		tempLeg[0]:=legExtendRefPosCurling[i,0];tempLeg[1]:=legExtendRefPosCurling[i,1];tempLeg[2]:=legExtendRefPosCurling[i,2];
		tempRef[0]:=jntExtendRefPosCurling[i,0];tempRef[1]:=jntExtendRefPosCurling[i,1];tempRef[2]:=jntExtendRefPosCurling[i,2];
		GVL.legCtrl[i].InverseKinetics(tipPosition:=tempLeg , refPosLast:=tempRef , legIndex:=i , motorAngles=>tempJnt , isSingular=> );
		jntAngExtend[i,0]:=tempJnt[0];jntAngExtend[i,1]:=tempJnt[1];jntAngExtend[i,2]:=tempJnt[2];			
		
	END_FOR
	tipForceDesire:=tipForceDesireZeros;

END_IF

IF RecoveryFinished=FALSE THEN
	body_ref_pos:=body_ref_pos_enter;
	body_ref_ang:=body_ref_ang_enter;
	leg_ref_pos:=leg_ref_pos_enter;
	
	IF (gait_cycle-EnterRecoveryCount)<=(tRetract + tWait + tExtend) * gvl.sampleRate THEN //leg 0-2-4 recovery
		
		//force compensator****************************
		IF (gait_cycle-EnterRecoveryCount)<=fceLoadTime*gvl.sampleRate THEN
			tr  := UDINT_TO_LREAL(gait_cycle-EnterRecoveryCount) / gvl.sampleRate /fceLoadTime;
			fbGetPivot(tNow := tr, tTotal := 1.0, pivot => pvt);
			FOR i:=0 TO 5 DO
				FOR j:=0 TO 2 DO
					tipForceDesire[i,j]:=(1-pvt)*tipForceDesireZeros[i,j]+pvt*tipForceDesireGroupB[i,j];//group B add load
				END_FOR
			END_FOR
		ELSIF  (gait_cycle-EnterRecoveryCount)>LREAL_TO_UDINT((tRetract + tWait + tExtend-fceLoadTime)*gvl.sampleRate) AND  (gait_cycle-EnterRecoveryCount)<=LREAL_TO_UDINT((tRetract + tWait + tExtend) * gvl.sampleRate) THEN
			tr  := (UDINT_TO_LREAL (gait_cycle-EnterRecoveryCount) / gvl.sampleRate-(tRetract + tWait + tExtend-fceLoadTime) )/fceLoadTime;
			fbGetPivot(tNow := tr, tTotal := 1.0, pivot => pvt);
			FOR i:=0 TO 5 BY 2DO
				FOR j:=0 TO 2 DO
					//tipForceDesire[i,j]:=(1-pvt)*tipForceDesireZeros[i,j]+pvt*tipForceDesireGroupA[i,j];//group A add load
					tipForceDesire[i+1,j]:=(1-pvt)*tipForceDesireGroupB[i+1,j]+pvt*tipForceDesireZeros[i+1,j];//group B reduce load
				END_FOR
			END_FOR
		ELSE
		tipForceDesire:=tipForceDesireGroupB;
		END_IF
		//***********************************************
	
		IF gait_cycle-EnterRecoveryCount < tRetract * gvl.sampleRate THEN
			tTotal := tRetract;
			tNow   := UDINT_TO_LREAL(gait_cycle-EnterRecoveryCount) * 1.0 / DINT_TO_LREAL(gvl.sampleRate);
			jntPosBegin := RcJointPosStart;
			FOR i:=0 TO 5 BY 2 DO
				FOR j:=0 TO 2 DO
					jntPosEnd[i,j]:=jntAngRetract[i,j];
					jntPosEnd[i+1,j]:=RcJointPosStart[i+1,j];
				END_FOR
			END_FOR
		ELSIF gait_cycle-EnterRecoveryCount  < (tRetract + tWait) * gvl.sampleRate THEN
			tTotal := tWait;
			tNow   := UDINT_TO_LREAL(gait_cycle-EnterRecoveryCount) * 1.0 / DINT_TO_LREAL(gvl.sampleRate) - tRetract;
			FOR i:=0 TO 5 BY 2 DO
				FOR j:=0 TO 2 DO
					jntPosBegin[i,j]:=jntAngRetract[i,j];
					jntPosBegin[i+1,j]:=RcJointPosStart[i+1,j];
					jntPosEnd[i,j]:=jntAngRetract[i,j];
					jntPosEnd[i+1,j]:=RcJointPosStart[i+1,j];
				END_FOR
			END_FOR
		ELSE 
			tTotal := tExtend;
			tNow   := UDINT_TO_LREAL(gait_cycle-EnterRecoveryCount) * 1.0 / DINT_TO_LREAL(gvl.sampleRate) - tRetract - tWait;
			FOR i:=0 TO 5 BY 2 DO
				FOR j:=0 TO 2 DO
					jntPosBegin[i,j]:=jntAngRetract[i,j];
					jntPosBegin[i+1,j]:=RcJointPosStart[i+1,j];
					jntPosEnd[i,j]:=jntAngExtend[i,j];
					jntPosEnd[i+1,j]:=RcJointPosStart[i+1,j];
				END_FOR
			END_FOR	
		END_IF	
	ELSIF (gait_cycle-EnterRecoveryCount)<=2*(tRetract + tWait + tExtend) * gvl.sampleRate  THEN //leg 1-3-5 recovery

		//force compensator*******************
		IF (gait_cycle-EnterRecoveryCount)>LREAL_TO_UDINT((tRetract + tWait + tExtend)*gvl.sampleRate) AND (gait_cycle-EnterRecoveryCount)<=LREAL_TO_UDINT((tRetract + tWait + tExtend+fceLoadTime)* gvl.sampleRate) THEN
			tr  := (UDINT_TO_LREAL(gait_cycle-EnterRecoveryCount) / gvl.sampleRate-(tRetract + tWait + tExtend) )/fceLoadTime;
			fbGetPivot(tNow := tr, tTotal := 1.0, pivot => pvt);
			FOR i:=0 TO 5 BY 2 DO
				FOR j:=0 TO 2 DO
					tipForceDesire[i,j]:=(1-pvt)*tipForceDesireZeros[i,j]+pvt*tipForceDesireGroupA[i,j];//group A add load
					tipForceDesire[i+1,j]:=tipForceDesireZeros[i+1,j];//group B zeros load
				END_FOR
			END_FOR		
		ELSIF (gait_cycle-EnterRecoveryCount)>LREAL_TO_UDINT((2*(tRetract + tWait + tExtend)-fceLoadTime)*gvl.sampleRate) AND (gait_cycle-EnterRecoveryCount)<=LREAL_TO_UDINT(2*(tRetract + tWait + tExtend) * gvl.sampleRate) THEN
			tr  := (UDINT_TO_LREAL(gait_cycle-EnterRecoveryCount) / gvl.sampleRate-(2*(tRetract + tWait + tExtend)-fceLoadTime) )/fceLoadTime;
			fbGetPivot(tNow := tr, tTotal := 1.0, pivot => pvt);
			FOR i:=0 TO 5 BY 2DO
				FOR j:=0 TO 2 DO
					tipForceDesire[i,j]:=(1-pvt)*tipForceDesireGroupA[i,j]+pvt*tipForceDesireZeros[i,j];//group A reduce load
					tipForceDesire[i+1,j]:=tipForceDesireZeros[i+1,j];//group B zeros load
				END_FOR
			END_FOR	
		ELSE	
			tipForceDesire:=tipForceDesireGroupA;
		END_IF	
		//******************************************	

		
		IF gait_cycle-EnterRecoveryCount<=(2*tRetract + tWait + tExtend) * gvl.sampleRate THEN
			tTotal := tRetract;
			tNow   := UDINT_TO_LREAL(gait_cycle-EnterRecoveryCount) * 1.0 / DINT_TO_LREAL(gvl.sampleRate)-(tRetract + tWait + tExtend);
			FOR i:=0 TO 5 BY 2 DO
				FOR j:=0 TO 2 DO
					jntPosBegin[i,j]:=jntAngExtend[i,j];
					jntPosBegin[i+1,j]:=RcJointPosStart[i+1,j];
					jntPosEnd[i,j]:=jntAngExtend[i,j];
					jntPosEnd[i+1,j]:=jntAngRetract[i+1,j];
				END_FOR
			END_FOR			
		ELSIF gait_cycle-EnterRecoveryCount<=(2*tRetract + 2*tWait + tExtend) * gvl.sampleRate THEN
			tTotal := tWait;
			tNow   := UDINT_TO_LREAL(gait_cycle-EnterRecoveryCount) * 1.0 / DINT_TO_LREAL(gvl.sampleRate) - (2*tRetract + tWait + tExtend);
			FOR i:=0 TO 5 BY 2 DO
				FOR j:=0 TO 2 DO
					jntPosBegin[i,j]:=jntAngExtend[i,j];
					jntPosBegin[i+1,j]:=jntAngRetract[i+1,j];
					jntPosEnd[i,j]:=jntAngExtend[i,j];
					jntPosEnd[i+1,j]:=jntAngRetract[i+1,j];
				END_FOR
			END_FOR			
		ELSE
			tTotal := tExtend;
			tNow   := UDINT_TO_LREAL(gait_cycle-EnterRecoveryCount) * 1.0 / DINT_TO_LREAL(gvl.sampleRate) - (2*tRetract + 2*tWait + tExtend);
			FOR i:=0 TO 5 BY 2 DO
				FOR j:=0 TO 2 DO
					jntPosBegin[i,j]:=jntAngExtend[i,j];
					jntPosBegin[i+1,j]:=jntAngRetract[i+1,j];
					jntPosEnd[i,j]:=jntAngExtend[i,j];
					jntPosEnd[i+1,j]:=jntAngExtend[i+1,j];
				END_FOR
			END_FOR			
		END_IF
	ELSE
		tTotal := 100;
		tNow   := UDINT_TO_LREAL(gait_cycle-EnterRecoveryCount) * 1.0 / DINT_TO_LREAL(gvl.sampleRate) - 2*tRetract - 2*tWait - 2*tExtend;
		jntPosBegin :=jntAngExtend;
		jntPosEnd :=jntAngExtend;
		RecoveryFinished:=TRUE;
		tipForceDesire:=tipForceDesireZeros;
	END_IF
	getPivot(tNow := tNow, tTotal := tTotal, pivot => pivot, pivotDot => pivotDot);
	FOR i := 0 TO 5 DO
		FOR j := 0 TO 2 DO
			RcJointPosRef[i, j] := (1.0 - pivot) * jntPosBegin[i, j] + pivot * jntPosEnd[i, j];
		END_FOR
		tempJnt[0]:=RcJointPosRef[i,0];tempJnt[1]:=RcJointPosRef[i,1];tempJnt[2]:=RcJointPosRef[i,2];
		gvl.legCtrl[i].ForwardKinetics(motorAngles:=tempJnt , legIndex:=i , tipPosition=>Rc_PosWrtHip[i].data );
		fbRotMat(yaw := body_ref_ang_enter.data[2], pitch := body_ref_ang_enter.data[1],roll := body_ref_ang_enter.data[0], rm =>  Rb_target1 );
		temp.data[0]:=hip_pos[i,0];temp.data[1]:=hip_pos[i,1];temp.data[2]:=hip_pos[i,2];
		leg_ref_pos[i]:= VecAdd( MatMulVec(Rb_target1, VecAdd(temp,MatMulVec(Rleg[i],Rc_PosWrtHip[i]))),body_ref_pos);		
	END_FOR

END_IF
END_METHOD

METHOD PUBLIC TrjPlanning_SearchPedal : BOOL
VAR_INPUT
END_VAR
VAR
	tr: LREAL;
	i: INT;
	j: INT;
	Rb_target1: Mat3;
	temp: vec3;
	
	tipForceDesireLegA:	 ARRAY[0..5,0..2] OF LREAL:=[0,-100,0,
													 0,0,0,
													 0,0,0,
													 0,0,0,
													 0,0,0,
													 0,0,0];
	tipForceDesireLegF:	 ARRAY[0..5,0..2] OF LREAL:=[0,0,0,
													 0,0,0,
													 0,0,0,
													 0,0,0,
													 0,0,0,
													 0,-120,0];				
END_VAR
IF SearchPedalFinished=FALSE THEN
	IF SP_RBLegSearching=TRUE THEN
		SP_LBLegSearching:=FALSE;
		body_ref_pos:=body_ref_pos_enter;
		body_ref_ang:=body_ref_ang_enter;
		leg_ref_pos:=leg_ref_pos_enter;	
		IF (gait_cycle-SP_EnterSubSearchCount[0])<=SP_LiftLegTime*gvl.sampleRate THEN
			tr  := UDINT_TO_LREAL(gait_cycle - SP_EnterSubSearchCount[0]) / gvl.sampleRate / SP_LiftLegTime;
			fbGetPivot(tNow := tr, tTotal := 1.0, pivot => pvt);	
			SP_BPosRefWrtHip[0].data[0]:=SP_BPosStartWrtHip[0].data[0];
			SP_BPosRefWrtHip[0].data[1]:=(1-pvt)*SP_BPosStartWrtHip[0].data[1]+pvt*(SP_BPosStartWrtHip[0].data[1]+SP_LiftDistance);
			SP_BPosRefWrtHip[0].data[2]:=SP_BPosStartWrtHip[0].data[2];
			fbRotMat(yaw := body_ref_ang_enter.data[2], pitch := body_ref_ang_enter.data[1],roll := body_ref_ang_enter.data[0], rm =>  Rb_target1 );
			temp.data[0]:=hip_pos[0,0];temp.data[1]:=hip_pos[0,1];temp.data[2]:=hip_pos[0,2];
			leg_ref_pos[0]:= VecAdd( MatMulVec(Rb_target1, VecAdd(temp,MatMulVec(Rleg[0],SP_BPosRefWrtHip[0]))),body_ref_pos);	
			
			//force compensator
			tipForceTarget:=tipForceDesireLegF;
			IF (gait_cycle-SP_EnterSubSearchCount[0])<=LREAL_TO_UDINT(fceLoadTime*gvl.sampleRate) THEN
				tr  := (UDINT_TO_LREAL(gait_cycle-SP_EnterSubSearchCount[0]) / gvl.sampleRate)/ fceLoadTime;
				fbGetPivot(tNow := tr, tTotal := 1.0, pivot => pvt);
				FOR i:=0 TO 5 DO
					FOR j:=0 TO 2 DO
						tipForceDesire[i,j]:=(1-pvt)*tipForceDesireZeros[i,j]+pvt*tipForceTarget[i,j];
					END_FOR
				END_FOR
			END_IF
			
		ELSIF (gait_cycle-SP_EnterSubSearchCount[0])<=(SP_LiftLegTime+SP_SearchTime)*gvl.sampleRate AND  SP_BLegSearchFinished[0]=FALSE THEN
			tr  := (UDINT_TO_LREAL(gait_cycle - SP_EnterSubSearchCount[0]) / gvl.sampleRate -SP_LiftLegTime)/ SP_SearchTime;
			fbGetPivot(tNow := tr, tTotal := 1.0, pivot => pvt);	
			SP_BPosRefWrtHip[0].data[0]:=(1-pvt)*SP_BPosStartWrtHip[0].data[0]+pvt*(SP_BPosStartWrtHip[0].data[0]-SP_SearchDistance);		
			SP_BPosRefWrtHip[0].data[1]:=SP_BPosStartWrtHip[0].data[1]+SP_LiftDistance;
			SP_BPosRefWrtHip[0].data[2]:=SP_BPosStartWrtHip[0].data[2];
			IF isPedal(0)=TRUE AND  SP_BLegSearchFinished[0]=FALSE THEN
				SP_BLegSearchFinished[0]:=TRUE;
				SP_EnterSubSearchDecreaseCount[0]:=gait_cycle;
				FOR j:=0 TO 2 DO
					SP_BPosLockWrtHip[0].data[j]:=SP_BPosRefWrtHip[0].data[j];
				END_FOR			
			END_IF
			IF (gait_cycle-SP_EnterSubSearchCount[0])=LREAL_TO_UDINT((SP_LiftLegTime+SP_SearchTime)*gvl.sampleRate) AND SP_BLegSearchFinished[0]=FALSE THEN
				SP_BLegSearchFinished[0]:=TRUE;
				SP_EnterSubSearchDecreaseCount[0]:=gait_cycle;
				FOR j:=0 TO 2 DO
					SP_BPosLockWrtHip[0].data[j]:=SP_BPosRefWrtHip[0].data[j];
				END_FOR	
			END_IF

			fbRotMat(yaw := body_ref_ang_enter.data[2], pitch := body_ref_ang_enter.data[1],roll := body_ref_ang_enter.data[0], rm =>  Rb_target1 );
			temp.data[0]:=hip_pos[0,0];temp.data[1]:=hip_pos[0,1];temp.data[2]:=hip_pos[0,2];
			leg_ref_pos[0]:= VecAdd( MatMulVec(Rb_target1, VecAdd(temp,MatMulVec(Rleg[0],SP_BPosRefWrtHip[0]))),body_ref_pos);	
			
		ELSIF  SP_BLegSearchFinished[0]=TRUE AND (gait_cycle-SP_EnterSubSearchDecreaseCount[0])<=SP_LiftLegTime*gvl.sampleRate THEN
			tr  := UDINT_TO_LREAL(gait_cycle - SP_EnterSubSearchDecreaseCount[0]) / gvl.sampleRate / SP_LiftLegTime;
			fbGetPivot(tNow := tr, tTotal := 1.0, pivot => pvt);
			SP_BPosRefWrtHip[0].data[0]:=SP_BPosLockWrtHip[0].data[0];	
			SP_BPosRefWrtHip[0].data[1]:=(1-pvt)*SP_BPosLockWrtHip[0].data[1]+pvt*(SP_BPosLockWrtHip[0].data[1]-SP_LiftDistance);
			SP_BPosRefWrtHip[0].data[2]:=SP_BPosLockWrtHip[0].data[2];	
			
			fbRotMat(yaw := body_ref_ang_enter.data[2], pitch := body_ref_ang_enter.data[1],roll := body_ref_ang_enter.data[0], rm =>  Rb_target1 );
			temp.data[0]:=hip_pos[0,0];temp.data[1]:=hip_pos[0,1];temp.data[2]:=hip_pos[0,2];
			leg_ref_pos[0]:= VecAdd( MatMulVec(Rb_target1, VecAdd(temp,MatMulVec(Rleg[0],SP_BPosRefWrtHip[0]))),body_ref_pos);	
			IF (gait_cycle-SP_EnterSubSearchDecreaseCount[0])=LREAL_TO_UDINT( SP_LiftLegTime*gvl.sampleRate) THEN
				body_ref_pos_enter:=body_ref_pos;
				body_ref_ang_enter:=body_ref_ang;
				leg_ref_pos_enter:=leg_ref_pos;	
			END_IF	
			
			//force compensator
			tipForceTarget:=tipForceDesireLegF;
			IF (gait_cycle-SP_EnterSubSearchDecreaseCount[0])>LREAL_TO_UDINT((SP_LiftLegTime-fceLoadTime)*gvl.sampleRate)THEN
				tr  := (UDINT_TO_LREAL(gait_cycle-SP_EnterSubSearchDecreaseCount[0]) / gvl.sampleRate-(SP_LiftLegTime-fceLoadTime) )/ fceLoadTime;
				fbGetPivot(tNow := tr, tTotal := 1.0, pivot => pvt);
				FOR i:=0 TO 5 DO
					FOR j:=0 TO 2 DO
						tipForceDesire[i,j]:=(1-pvt)*tipForceTarget[i,j]+pvt*tipForceDesireZeros[i,j];
					END_FOR
				END_FOR
			END_IF
	
		ELSE
			SP_RBLegSearching:=FALSE;
			SP_LBLegSearching:=TRUE;
			SP_EnterSubSearchCount[1]:=gait_cycle;			
		END_IF
	END_IF
	
	IF SP_LBLegSearching=TRUE THEN
		SP_RBLegSearching:=FALSE;
		body_ref_pos:=body_ref_pos_enter;
		body_ref_ang:=body_ref_ang_enter;
		leg_ref_pos:=leg_ref_pos_enter;	
		IF (gait_cycle-SP_EnterSubSearchCount[1])<=SP_LiftLegTime*gvl.sampleRate THEN
			tr  := UDINT_TO_LREAL(gait_cycle - SP_EnterSubSearchCount[1]) / gvl.sampleRate / SP_LiftLegTime;
			fbGetPivot(tNow := tr, tTotal := 1.0, pivot => pvt);	
			SP_BPosRefWrtHip[1].data[0]:=SP_BPosStartWrtHip[1].data[0];
			SP_BPosRefWrtHip[1].data[1]:=(1-pvt)*SP_BPosStartWrtHip[1].data[1]+pvt*(SP_BPosStartWrtHip[1].data[1]+SP_LiftDistance);
			SP_BPosRefWrtHip[1].data[2]:=SP_BPosStartWrtHip[1].data[2];
			fbRotMat(yaw := body_ref_ang_enter.data[2], pitch := body_ref_ang_enter.data[1],roll := body_ref_ang_enter.data[0], rm =>  Rb_target1 );
			temp.data[0]:=hip_pos[5,0];temp.data[1]:=hip_pos[5,1];temp.data[2]:=hip_pos[5,2];
			leg_ref_pos[5]:= VecAdd( MatMulVec(Rb_target1, VecAdd(temp,MatMulVec(Rleg[5],SP_BPosRefWrtHip[1]))),body_ref_pos);	
			
			//force compensator
			tipForceTarget:=tipForceDesireLegA;
			IF (gait_cycle-SP_EnterSubSearchCount[1])<=LREAL_TO_UDINT(fceLoadTime*gvl.sampleRate) THEN
				tr  := (UDINT_TO_LREAL(gait_cycle-SP_EnterSubSearchCount[1]) / gvl.sampleRate)/ fceLoadTime;
				fbGetPivot(tNow := tr, tTotal := 1.0, pivot => pvt);
				FOR i:=0 TO 5 DO
					FOR j:=0 TO 2 DO
						tipForceDesire[i,j]:=(1-pvt)*tipForceDesireZeros[i,j]+pvt*tipForceTarget[i,j];
					END_FOR
				END_FOR
			END_IF
			
		ELSIF (gait_cycle-SP_EnterSubSearchCount[1])<=(SP_LiftLegTime+SP_SearchTime)*gvl.sampleRate AND  SP_BLegSearchFinished[1]=FALSE THEN
			tr  := (UDINT_TO_LREAL(gait_cycle - SP_EnterSubSearchCount[1]) / gvl.sampleRate -SP_LiftLegTime)/ SP_SearchTime;
			fbGetPivot(tNow := tr, tTotal := 1.0, pivot => pvt);	
			SP_BPosRefWrtHip[1].data[0]:=(1-pvt)*SP_BPosStartWrtHip[1].data[0]+pvt*(SP_BPosStartWrtHip[1].data[0]-SP_SearchDistance);		
			SP_BPosRefWrtHip[1].data[1]:=SP_BPosStartWrtHip[1].data[1]+SP_LiftDistance;
			SP_BPosRefWrtHip[1].data[2]:=SP_BPosStartWrtHip[1].data[2];
			IF isPedal(5)=TRUE AND  SP_BLegSearchFinished[1]=FALSE THEN
				SP_BLegSearchFinished[1]:=TRUE;
				SP_EnterSubSearchDecreaseCount[1]:=gait_cycle;
				FOR j:=0 TO 2 DO
					SP_BPosLockWrtHip[1].data[j]:=SP_BPosRefWrtHip[1].data[j];
				END_FOR			
			END_IF
			IF (gait_cycle-SP_EnterSubSearchCount[1])=LREAL_TO_UDINT((SP_LiftLegTime+SP_SearchTime)*gvl.sampleRate) AND SP_BLegSearchFinished[1]=FALSE THEN
				SP_BLegSearchFinished[1]:=TRUE;
				SP_EnterSubSearchDecreaseCount[1]:=gait_cycle;
				FOR j:=0 TO 2 DO
					SP_BPosLockWrtHip[1].data[j]:=SP_BPosRefWrtHip[1].data[j];
				END_FOR	
			END_IF

			fbRotMat(yaw := body_ref_ang_enter.data[2], pitch := body_ref_ang_enter.data[1],roll := body_ref_ang_enter.data[0], rm =>  Rb_target1 );
			temp.data[0]:=hip_pos[5,0];temp.data[1]:=hip_pos[5,1];temp.data[2]:=hip_pos[5,2];
			leg_ref_pos[5]:= VecAdd( MatMulVec(Rb_target1, VecAdd(temp,MatMulVec(Rleg[5],SP_BPosRefWrtHip[1]))),body_ref_pos);	
			
		ELSIF  SP_BLegSearchFinished[1]=TRUE AND (gait_cycle-SP_EnterSubSearchDecreaseCount[1])<=SP_LiftLegTime*gvl.sampleRate THEN
			tr  := UDINT_TO_LREAL(gait_cycle - SP_EnterSubSearchDecreaseCount[1]) / gvl.sampleRate / SP_LiftLegTime;
			fbGetPivot(tNow := tr, tTotal := 1.0, pivot => pvt);
			SP_BPosRefWrtHip[1].data[0]:=SP_BPosLockWrtHip[1].data[0];	
			SP_BPosRefWrtHip[1].data[1]:=(1-pvt)*SP_BPosLockWrtHip[1].data[1]+pvt*(SP_BPosLockWrtHip[1].data[1]-SP_LiftDistance);
			SP_BPosRefWrtHip[1].data[2]:=SP_BPosLockWrtHip[1].data[2];	
			
			fbRotMat(yaw := body_ref_ang_enter.data[2], pitch := body_ref_ang_enter.data[1],roll := body_ref_ang_enter.data[0], rm =>  Rb_target1 );
			temp.data[0]:=hip_pos[5,0];temp.data[1]:=hip_pos[5,1];temp.data[2]:=hip_pos[5,2];
			leg_ref_pos[5]:= VecAdd( MatMulVec(Rb_target1, VecAdd(temp,MatMulVec(Rleg[5],SP_BPosRefWrtHip[1]))),body_ref_pos);	
			IF (gait_cycle-SP_EnterSubSearchDecreaseCount[1])=LREAL_TO_UDINT( SP_LiftLegTime*gvl.sampleRate) THEN
				body_ref_pos_enter:=body_ref_pos;
				body_ref_ang_enter:=body_ref_ang;
				leg_ref_pos_enter:=leg_ref_pos;	
			END_IF	
			
			//force compensator
			tipForceTarget:=tipForceDesireLegA;
			IF (gait_cycle-SP_EnterSubSearchDecreaseCount[1])>LREAL_TO_UDINT((SP_LiftLegTime-fceLoadTime)*gvl.sampleRate)THEN
				tr  := (UDINT_TO_LREAL(gait_cycle-SP_EnterSubSearchDecreaseCount[1]) / gvl.sampleRate-(SP_LiftLegTime-fceLoadTime) )/ fceLoadTime;
				fbGetPivot(tNow := tr, tTotal := 1.0, pivot => pvt);
				FOR i:=0 TO 5 DO
					FOR j:=0 TO 2 DO
						tipForceDesire[i,j]:=(1-pvt)*tipForceTarget[i,j]+pvt*tipForceDesireZeros[i,j];
					END_FOR
				END_FOR
			END_IF			
			
		ELSE
			SP_RBLegSearching:=FALSE;
			SP_LBLegSearching:=FALSE;	
			SearchPedalFinished:=TRUE;	
			tipForceDesire:=tipForceDesireZeros;
		END_IF
	END_IF	
END_IF
END_METHOD

METHOD PUBLIC TrjPlanning_Slide : BOOL
VAR_INPUT
END_VAR
IF SlideFinished=FALSE THEN
	body_ref_pos:=body_ref_pos_enter;
	body_ref_ang:=body_ref_ang_enter;
	leg_ref_pos:=leg_ref_pos_enter;

END_IF

//***********tuning***************************
IF SlideFinished=FALSE AND (gait_cycle-EnterSlideCount)>=LREAL_TO_UDINT(slideTime*gvl.sampleRate) THEN
	RequirePushReleaseBall:=TRUE;
END_IF

//*************end-tuning********************



IF SlideFinished=FALSE AND RequirePushReleaseBall=TRUE THEN
	SlideFinished:=TRUE;
END_IF
END_METHOD

METHOD PUBLIC TrjPlanning_SpeedDown : BOOL
VAR_INPUT
END_VAR

VAR
	tr: LREAL;
	i: INT;
	SpeedDown_MPosTarget:ARRAY[0..1,0..2] OF LREAL:=[-0.0141,-0.1797,-0.1246,
                                                        -0.0141,-0.1797,0.1246];
	SpeedDown_MJntTargetRef:ARRAY[0..1,0..2] OF LREAL:=[0,331.45*pi/180,-144*pi/180,
                                                     0,331.45*pi/180,-144*pi/180];
	j: INT;
	Rb_target1: Mat3;
	temp: vec3;
	tempLeg:ARRAY [0..2] OF LREAL;
	tempJnt:ARRAY [0..2] OF LREAL;
	tempRef:ARRAY [0..2] OF LREAL;
END_VAR
IF (gait_cycle-EnterSpeedDownCount)=1 THEN
	FOR i:=0 TO 1 DO
		tempLeg[0]:=SpeedDown_MPosTarget[i,0];tempLeg[1]:=SpeedDown_MPosTarget[i,1];tempLeg[2]:=SpeedDown_MPosTarget[i,2];
		tempRef[0]:=SpeedDown_MJntTargetRef[i,0];tempRef[1]:=SpeedDown_MJntTargetRef[i,1];tempRef[2]:=SpeedDown_MJntTargetRef[i,2];
		GVL.legCtrl[Mapping14[i]].InverseKinetics(tipPosition:=tempLeg , refPosLast:=tempRef , legIndex:=Mapping14[i] , motorAngles=>tempJnt , isSingular=> );
		SpeedDown_MJntTarget[i,0]:=tempJnt[0];SpeedDown_MJntTarget[i,1]:=tempJnt[1];SpeedDown_MJntTarget[i,2]:=tempJnt[2];		
	END_FOR
END_IF

IF SpeedDownFinished=FALSE THEN
	IF gait_cycle-EnterSpeedDownCount<=SpeedDownTime*gvl.sampleRate THEN
		body_ref_pos:=body_ref_pos_enter;
		body_ref_ang:=body_ref_ang_enter;
		leg_ref_pos:=leg_ref_pos_enter;
		tr  := UDINT_TO_LREAL(gait_cycle - EnterSpeedDownCount) / gvl.sampleRate / SpeedDownTime;
		fbGetPivot(tNow := tr, tTotal := 1.0, pivot => pvt);
		FOR i:=0 TO 1 DO
			FOR j:=0 TO 2 DO
				SpeedDown_MJntRef[i].data[j]:=(1-pvt)*SpeedDown_MJntStart[i].data[j]+pvt*SpeedDown_MJntTarget[i,j];
			END_FOR
			gvl.legCtrl[Mapping14[i]].ForwardKinetics(motorAngles:=SpeedDown_MJntRef[i].data , legIndex:=Mapping14[i] , tipPosition=>SpeedDown_MPosWrtHip[i].data );
			fbRotMat(yaw := body_ref_ang_enter.data[2], pitch := body_ref_ang_enter.data[1],roll := body_ref_ang_enter.data[0], rm =>  Rb_target1 );
			temp.data[0]:=hip_pos[Mapping14[i],0];temp.data[1]:=hip_pos[Mapping14[i],1];temp.data[2]:=hip_pos[Mapping14[i],2];
			leg_ref_pos[Mapping14[i]]:= VecAdd( MatMulVec(Rb_target1, VecAdd(temp,MatMulVec(Rleg[Mapping14[i]],SpeedDown_MPosWrtHip[i]))),body_ref_pos);
			
			leg_ref_pos[Mapping05[i]].data[2]:=(1-pvt)*leg_ref_pos_enter[Mapping05[i]].data[2]+pvt*(leg_ref_pos_enter[Mapping05[i]].data[2]-Distance_y_DS-0.005);
		END_FOR
	ELSE
		SpeedDownFinished:=TRUE;
	END_IF
	
	IF gait_cycle-EnterSpeedDownCount=1 THEN
		GVL.jogVelocity[18]:=0;
		GVL.jogVelocity[19]:=0;
		gvl.jogStopButton[18]:=TRUE;
		gvl.jogStopButton[19]:=TRUE;
		gvl.motorDrive[j].SetTrgVel(0);
	END_IF
END_IF
END_METHOD

METHOD PUBLIC TrjPlanning_SpeedUp : BOOL
VAR_INPUT
END_VAR

VAR
	invalid: LREAL;
	Rb_target1: Mat3;
	i: INT;
	tr: LREAL;
	temp: VEC3;
	
	
	tipForceDesireLegAF:	 ARRAY[0..5,0..2] OF LREAL:=[0,-30,0,
													 0,0,0,
													 0,0,0,
													 0,0,0,
													 0,0,0,
													 0,-30,0];
	j: INT;
END_VAR
IF SpeedUpSubState=SpeedUpAS AND (gait_cycle-EnterSpeedUpASCount)=LREAL_TO_UDINT(Time_AS*gvl.sampleRate) THEN
	SpeedUpSubState:=SpeedUpCS;
	EnterSpeedUpCSCount:=gait_cycle;
	body_ref_pos_enter :=body_ref_pos;
	body_ref_ang_enter:=body_ref_ang;
	leg_ref_pos_enter := leg_ref_pos;
	
ELSIF SpeedUpSubState=SpeedUpCS AND gait_cycle-EnterSpeedUpCSCount=LREAL_TO_UDINT(Time_CS*gvl.sampleRate) THEN
	SpeedUpSubState:=SpeedUpDS;
	EnterSpeedUpDSCount:=gait_cycle;
	body_ref_pos_enter :=body_ref_pos;
	body_ref_ang_enter:=body_ref_ang;
	leg_ref_pos_enter := leg_ref_pos;
ELSIF SpeedUpSubState=SpeedUpDS AND gait_cycle-EnterSpeedUpDSCount=LREAL_TO_UDINT(Time_DS*gvl.sampleRate) THEN
	SpeedUpSubState:=SpeedUpSS;
	EnterSpeedUpSPCount:=gait_cycle;
	body_ref_pos_enter :=body_ref_pos;
	body_ref_ang_enter:=body_ref_ang;
	leg_ref_pos_enter := leg_ref_pos;
	SpeedUpFinished:=TRUE;
	tipForceDesire:=tipForceDesireZeros;
	RequireSlide:=TRUE;
END_IF

body_ref_pos:=body_ref_pos_enter;
body_ref_ang:=body_ref_ang_enter;
leg_ref_pos:=leg_ref_pos_enter;

IF SpeedUpSubState=SpeedUpAS AND gait_cycle-EnterSpeedUpASCount<=Time_AS*gvl.sampleRate THEN
	fbHermitInterpolation(t0:=EnterSpeedUpASCount*delta_t , T:=Time_AS , y0:=0 , 
		y1:=Distance_x_AS , v0:=0 , v1:=target_vel , tNow:=gait_cycle* delta_t, 
		y=> body_ref_pos_wrt_body.data[0], v=>invalid );	
	body_ref_pos_wrt_body.data[1]:=0;body_ref_pos_wrt_body.data[2]:=0;
	fbRotMat(yaw := body_ref_ang_enter.data[2], pitch := body_ref_ang_enter.data[1],roll := body_ref_ang_enter.data[0], rm =>  Rb_target1 );
	body_ref_pos:=VecAdd(body_ref_pos_enter,MatMulVec(Rb_target1,body_ref_pos_wrt_body));
	
	//force compensator
	tipForceTarget:=tipForceDesireLegAF;
	IF (gait_cycle-EnterSpeedUpASCount)<=fceLoadTime*gvl.sampleRate THEN
		tr  := UDINT_TO_LREAL(gait_cycle-EnterSpeedUpASCount) / gvl.sampleRate / fceLoadTime;
		fbGetPivot(tNow := tr, tTotal := 1.0, pivot => pvt);
		FOR i:=0 TO 5 DO
			FOR j:=0 TO 2 DO
				tipForceDesire[i,j]:=(1-pvt)*tipForceDesireZeros[i,j]+pvt*tipForceTarget[i,j];
			END_FOR
		END_FOR	
	END_IF
	
END_IF
	//force compensator
	tipForceTarget:=tipForceDesireLegAF;
	IF (gait_cycle-EnterSpeedUpASCount)>(Time_AS+Time_CS-fceLoadTime)*gvl.sampleRate AND (gait_cycle-EnterSpeedUpASCount)<=(Time_AS+Time_CS)*gvl.sampleRate THEN
		tr  := (UDINT_TO_LREAL(gait_cycle-EnterSpeedUpASCount) / gvl.sampleRate- (Time_AS+Time_CS-fceLoadTime))/ fceLoadTime;
		fbGetPivot(tNow := tr, tTotal := 1.0, pivot => pvt);
		FOR i:=0 TO 5 DO
			FOR j:=0 TO 2 DO
				tipForceDesire[i,j]:=(1-pvt)*tipForceTarget[i,j]+pvt*tipForceDesireZeros[i,j];
			END_FOR
		END_FOR	
	END_IF

IF SpeedUpSubState=SpeedUpCS AND gait_cycle-EnterSpeedUpCSCount<=Time_CS*gvl.sampleRate THEN
	fbHermitInterpolation(t0:=EnterSpeedUpCSCount*delta_t , T:=Time_CS , y0:=0 , 
		y1:=target_vel*Time_CS , v0:=target_vel , v1:=target_vel , tNow:=gait_cycle* delta_t, 
		y=> body_ref_pos_wrt_body.data[0], v=>invalid );
	body_ref_pos_wrt_body.data[1]:=0;body_ref_pos_wrt_body.data[2]:=0;
	fbRotMat(yaw := body_ref_ang_enter.data[2], pitch := body_ref_ang_enter.data[1],roll := body_ref_ang_enter.data[0], rm =>  Rb_target1 );
	body_ref_pos:=VecAdd(body_ref_pos_enter,MatMulVec(Rb_target1,body_ref_pos_wrt_body));
END_IF
IF SpeedUpSubState=SpeedUpDS AND gait_cycle-EnterSpeedUpDSCount<=Time_DS*gvl.sampleRate THEN
	fbHermitInterpolation(t0:=EnterSpeedUpDSCount*delta_t , T:=Time_DS , y0:=0 , 
		y1:=Distance_x_DS , v0:=target_vel , v1:=0 , tNow:=gait_cycle* delta_t, 
		y=> body_ref_pos_wrt_body.data[0], v=>invalid );
	body_ref_pos_wrt_body.data[1]:=0;body_ref_pos_wrt_body.data[2]:=0;
	
	fbRotMat(yaw := body_ref_ang_enter.data[2], pitch := body_ref_ang_enter.data[1],roll := body_ref_ang_enter.data[0], rm =>  Rb_target1 );
	body_ref_pos:=VecAdd(body_ref_pos_enter,MatMulVec(Rb_target1,body_ref_pos_wrt_body));
	
	tr  := UDINT_TO_LREAL(gait_cycle - EnterSpeedUpDSCount) / gvl.sampleRate / Time_DS;
	fbGetPivot(tNow := tr, tTotal := 1.0, pivot => pvt);
	FOR i:=0 TO 1 DO
		leg_ref_pos[Mapping05[i]].data[2]:=(1-pvt)*leg_ref_pos_enter[Mapping05[i]].data[2]+pvt*(leg_ref_pos_enter[Mapping05[i]].data[2]+Distance_y_DS);
	END_FOR
	
END_IF
IF SpeedUpSubState=SpeedUpAS OR SpeedUpSubState=SpeedUpCS OR SpeedUpSubState=SpeedUpDS THEN
	FOR i:=0 TO 1 DO
		gvl.legCtrl[Mapping14[i]].ForwardKinetics(motorAngles:=SpeedUp_MJntRef[i].data , legIndex:=Mapping14[i] , tipPosition=>SpeedUp_MPosWrtHip[i].data );
		gvl.legCtrl[Mapping23[i]].ForwardKinetics(motorAngles:=SpeedUp_FJntRef[i].data , legIndex:=Mapping23[i] , tipPosition=>SpeedUp_FPosWrtHip[i].data );
		fbRotMat(yaw := body_ref_ang_enter.data[2], pitch := body_ref_ang_enter.data[1],roll := body_ref_ang_enter.data[0], rm =>  Rb_target1 );
		temp.data[0]:=hip_pos[Mapping14[i],0];temp.data[1]:=hip_pos[Mapping14[i],1];temp.data[2]:=hip_pos[Mapping14[i],2];
		leg_ref_pos[Mapping14[i]]:= VecAdd( MatMulVec(Rb_target1, VecAdd(temp,MatMulVec(Rleg[Mapping14[i]],SpeedUp_MPosWrtHip[i]))),body_ref_pos);
		temp.data[0]:=hip_pos[Mapping23[i],0];temp.data[1]:=hip_pos[Mapping23[i],1];temp.data[2]:=hip_pos[Mapping23[i],2];
		leg_ref_pos[Mapping23[i]]:= VecAdd( MatMulVec(Rb_target1, VecAdd(temp,MatMulVec(Rleg[Mapping23[i]],SpeedUp_FPosWrtHip[i]))),body_ref_pos);
	END_FOR
END_IF
END_METHOD

METHOD PUBLIC TrjPlanning_StoneRot : BOOL
VAR_INPUT
END_VAR
VAR
	(*StoneRot_FJntTarget:ARRAY[0..1,0..2] OF LREAL:=[-90*pi/180,524*pi/180,-190*pi/180,
                                                     90*pi/180,524*pi/180,-190*pi/180];*)
													 
	(*StoneRot_FJntTarget:ARRAY[0..1,0..2] OF LREAL:=[-90*pi/180,165*pi/180,(-190+360)*pi/180,
                                                     90*pi/180,165*pi/180,(-190+360)*pi/180];	//164 lose,165T 170S lose;*)
	StoneRot_FJntTarget:ARRAY[0..1,0..2] OF LREAL:=[-90*pi/180,167*pi/180,(171)*pi/180,
                                                     90*pi/180,167*pi/180,(171)*pi/180];	//164 lose,166T 168S passive wheels colide;												 
	tr: LREAL;
	i: INT;
	Rb_target1: Mat3;	
	temp:vec3;										 
	j: INT;
	noPlanning: BOOL;
END_VAR
//*****************************test trajectory*****************************************

	FOR i:=0 TO 1 DO
		(*IF SetColide=TRUE THEN
			gvl.tipActualFce[Mapping23[i],2]:=100;
		END_IF	*)
		(*IF(gait_cycle-EnterStoneRotCount)=0.5*StoneGripTime*gvl.sampleRate THEN
			gvl.tipActualFce[Mapping23[i],2]:=100;
		END_IF *)
		noPlanning:=TRUE;
	END_FOR
	

//**********************************end************************************************	

(*FOR i:=0 TO 1 DO
	IF StoneRotSubState[i]=FALSE AND isStone(Mapping23[i]) THEN
		StoneRotSubState[i]:=TRUE;
		leg_ref_pos_enter[Mapping23[i]]:=leg_ref_pos[Mapping23[i]];
	END_IF
END_FOR*)

IF (StoneRotSubState[0]=FALSE OR StoneRotSubState[1]=FALSE) AND (gait_cycle-EnterStoneRotCount)=LREAL_TO_UDINT(StoneGripTime*gvl.sampleRate) THEN
	StoneRotSubState[0]:=TRUE;
	StoneRotSubState[1]:=TRUE;
	leg_ref_pos_enter[Mapping23[0]]:=leg_ref_pos[Mapping23[0]];
	leg_ref_pos_enter[Mapping23[1]]:=leg_ref_pos[Mapping23[1]];
END_IF
	
body_ref_pos:=body_ref_pos_enter;
body_ref_ang:=body_ref_ang_enter;
leg_ref_pos:=leg_ref_pos_enter;


	IF (gait_cycle-EnterStoneRotCount)<=StoneGripTime*gvl.sampleRate THEN
		FOR i:=0 TO 1 DO
			IF StoneRotSubState[i]=FALSE THEN
			tr  := UDINT_TO_LREAL(gait_cycle - EnterStoneRotCount) / gvl.sampleRate /StoneGripTime;
			fbGetPivot(tNow := tr, tTotal := 1.0, pivot => pvt);
			FOR j:=0 TO 2 DO
				StoneRot_FJntRef[i].data[j]:=(1-pvt)*StoneRot_FJntStart[i].data[j]+pvt*(StoneRot_FJntTarget[i,j]);
			END_FOR
			gvl.legCtrl[Mapping23[i]].ForwardKinetics(motorAngles:=StoneRot_FJntRef[i].data , legIndex:=Mapping23[i] , tipPosition=>StoneRot_FPosWrtHip[i].data );
			fbRotMat(yaw := body_ref_ang_enter.data[2], pitch := body_ref_ang_enter.data[1],roll := body_ref_ang_enter.data[0], rm =>  Rb_target1 );
			temp.data[0]:=hip_pos[Mapping23[i],0];temp.data[1]:=hip_pos[Mapping23[i],1];temp.data[2]:=hip_pos[Mapping23[i],2];
			leg_ref_pos[Mapping23[i]]:= VecAdd( MatMulVec(Rb_target1, VecAdd(temp,MatMulVec(Rleg[Mapping23[i]],StoneRot_FPosWrtHip[i]))),body_ref_pos);
			END_IF
		END_FOR
	ELSE
		noPlanning:=TRUE;
	END_IF

IF (gait_cycle-EnterStoneRotCount)>StoneGripTime*gvl.sampleRate  THEN
		stone_rot_vel:=GVL.stone_rot_vel/60*2*pi;
		GVL.jogVelocity[18]:=stone_rot_vel;
		GVL.jogVelocity[19]:=-stone_rot_vel;
		FOR j:=18 TO 19 DO
			gvl.motorDrive[j].SetTrgVel(GVL.jogVelocity[j]);
			IF gvl.motorDrive[j].cvSetVel = GVL.jogVelocity[j] THEN
				gvl.jogButton[j]:=FALSE;
			ELSE
				gvl.jogButton[j]:=TRUE;
			END_IF
		END_FOR
END_IF

IF StoneRotFinished=FALSE AND (gait_cycle-EnterStoneRotCount)>=(StoneGripTime+StoneRotTime)*gvl.sampleRate THEN
	StoneRotFinished:=TRUE;
END_IF
END_METHOD

END_FUNCTION_BLOCK

(* stored: Version 1.1.0.1, ProductVersion 3.1.4024.2
   POU CurlingGaitFromSlip: Id {60870fbe-9372-4644-8201-6ee4a114d2cf}, SpecialFunc None
   Method DoPlanning: Id {a526c105-864a-4ef3-a646-bb7632c42b5f}
   Method Initialize: Id {9bdfb3b6-4c18-49e5-bc86-7a870e5fcc33}
   Method isPedal: Id {33785039-937e-483a-8149-9a6f9589866a}
   Method isStone: Id {3828978a-85ac-4eb4-8168-c31866fd1ac4}
   Method SetTargetValue: Id {e1935ec6-c32b-41cc-a62d-b61459b5fd30}
   Method StateMachine: Id {5ef4ea9d-f719-4140-9cda-9aefc2e8dc7a}
   Method TrjPlanning: Id {33080927-9d47-4eee-921a-6bb8a64b1112}
   Method TrjPlanning_AddHeight: Id {acb813a6-b8d3-446e-a4d2-e1b9c2cdd5b4}
   Method TrjPlanning_ArmControl: Id {99fa43a9-ec94-415c-9cd9-37ff750f7e87}
   Method TrjPlanning_BLegPosAdjust: Id {3093e979-b721-4bdb-95bd-ab44a7107aa5}
   Method TrjPlanning_BLegRecovery: Id {cd829a26-9eb0-4fd9-96d1-940c236395fe}
   Method TrjPlanning_BodyPosAdjust: Id {7f0117a2-a706-4595-9d97-7df79ab3b366}
   Method TrjPlanning_FlegRotB: Id {c1a7410f-1fb6-41d5-8519-4751dfebdb87}
   Method TrjPlanning_LiftMleg: Id {a543d1fd-a688-4e1e-a9a0-947506f19caf}
   Method TrjPlanning_MlegRollA: Id {bfb227bd-ca7c-4e4b-92fd-b1a2b93a0523}
   Method TrjPlanning_MlegRollB: Id {76260543-839c-4ac6-a04d-6f8340937b67}
   Method TrjPlanning_MlegRollC: Id {1efdfdee-aac4-4607-8bb9-71a9039f3b56}
   Method TrjPlanning_OrientAdjust: Id {c5614f0e-7d15-4bbe-abbe-5ce678ea12eb}
   Method TrjPlanning_PushReleaseBall: Id {7d1f3c30-c37f-4bad-b558-a2d3f42b8ebf}
   Method TrjPlanning_Recovery: Id {49cc427e-6f17-473f-b13a-91b056dab185}
   Method TrjPlanning_SearchPedal: Id {2846425e-3725-4c35-a469-4d40662ea1ed}
   Method TrjPlanning_Slide: Id {fd34b191-9e6b-4b9c-ae25-d126c0b1a096}
   Method TrjPlanning_SpeedDown: Id {81e2b8e0-3c72-4f11-ab88-0b0d07738684}
   Method TrjPlanning_SpeedUp: Id {ec3e324f-81e5-46b7-a74b-a5cc21d5d110}
   Method TrjPlanning_StoneRot: Id {34d2400a-79ce-4ff8-9998-c64a1e3d0b03} *)
